(*			
	RAFALOS
	Rafał Osajda		19.09.2025		TC 4024.66
	Element bazowy umożliwiający potomkom wysyłaś zgłoszenia do logera
*)
FUNCTION_BLOCK FB_BaseLoggerElement EXTENDS FB_Base IMPLEMENTS ITF_BaseLoggerElement, ITF_BaseLoggerElement_HMI_Connector
VAR
	itfLogger						: ITF_BaseLogger;
	stIdentifier					: ST_BaseElementIdentifier;
	stEvents						: ST_BaseEvents;
END_VAR

(*			
	EVERDE sp. z o.o.
	Rafał Osajda		24.03.2025		TC 4024.66
	Dodawanie zgłoszenia do systemu
*)
METHOD PUBLIC AddEvent : BOOL
VAR_INPUT
	bIgnoreRepetitions					: BOOL;						//jak true nie zliczaj powtorzeń wystapienia np komunikaty
	eEventCategory						: E_BaseEvents_Category;	//BYTE;	//1 - blad, 2 - ostrzezenie, 3 - wiadomosc, 4 - safety
	bConfirm							: BOOL;						//wymaga powtierdzenia
	stDescription						: ST_BaseLabel;
END_VAR
IF (THIS^.stEvents.uiNumberOfAdded + 1 <= GVL_BaseConstans.MAX_ILOSC_ZGLOSZEN_NA_ELEMENT) THEN
	THIS^.stEvents.uiNumberOfAdded														:= THIS^.stEvents.uiNumberOfAdded + 1;
	THIS^.stEvents.arrDefinitions [THIS^.stEvents.uiNumberOfAdded].uiIDInItem			:= THIS^.stEvents.uiNumberOfAdded;
	THIS^.stEvents.arrDefinitions [THIS^.stEvents.uiNumberOfAdded].bIgnoreRepetitions	:= bIgnoreRepetitions;
	THIS^.stEvents.arrDefinitions [THIS^.stEvents.uiNumberOfAdded].eEventCategory		:= eEventCategory;
	THIS^.stEvents.arrDefinitions [THIS^.stEvents.uiNumberOfAdded].stDescription		:= stDescription;
	THIS^.stEvents.arrDefinitions [THIS^.stEvents.uiNumberOfAdded].bConfirm				:= bConfirm;
	AddEvent						:= TRUE;
ELSE
	AddEvent						:= FALSE;
END_IF
END_METHOD

(*			
	EVERDE sp. z o.o.
	Rafał Osajda		24.03.2025		TC 4024.66
	Definicja nowego zgłoszenia
*)
METHOD PUBLIC EventsDefinition : BOOL
MEMSET (
	destAddr		:= ADR (THIS^.stEvents.arrDefinitions),
	fillByte		:= 0,
	n				:= SIZEOF (THIS^.stEvents.arrDefinitions)
);
THIS^.stEvents.uiNumberOfAdded	:= 0;
END_METHOD

(*			
	RAFALOS
	Rafał Osajda		25.09.2025		TC 4024.66
	Metoda wywoływana w pierwszym cyklu
*)
METHOD PUBLIC FirstCycle : BOOL
VAR_INPUT
END_VAR

FirstCycle				:= TRUE;
END_METHOD

METHOD PUBLIC GetCode : STRING
VAR_INPUT
END_VAR
GetCode			:= THIS^.stIdentifier.sCode;
END_METHOD

METHOD PUBLIC GetID : UINT
VAR_INPUT
END_VAR
GetID				:= THIS^.stIdentifier.uiID;
END_METHOD

METHOD PUBLIC GetIdentyfier : ST_BaseElementIdentifier
VAR_INPUT
END_VAR
GetIdentyfier				:= THIS^.stIdentifier;
END_METHOD

METHOD PUBLIC GetName : ST_BaseLabel
VAR_INPUT
END_VAR
GetName				:= THIS^.stIdentifier.stName;
END_METHOD

METHOD PUBLIC GetType : E_BaseElementType
VAR_INPUT
END_VAR
GetType				:= THIS^.stIdentifier.eType;
END_METHOD

METHOD PUBLIC SetCode
VAR_INPUT
	sCode							: STRING;
END_VAR
THIS^.stIdentifier.sCode				:= sCode;
END_METHOD

METHOD PUBLIC SetID
VAR_INPUT
	uiID					: UINT;
END_VAR
THIS^.stIdentifier.uiID			:= uiID;
END_METHOD

METHOD PUBLIC SetName
VAR_INPUT
	stName				: ST_BaseLabel;
END_VAR
this^.stIdentifier.stName			:= stName;
END_METHOD

METHOD PUBLIC SetType
VAR_INPUT
	eType					: E_BaseElementType;
END_VAR
THIS^.stIdentifier.eType				:= eType;
END_METHOD

END_FUNCTION_BLOCK

(* stored: Version 1.1.0.1
   POU FB_BaseLoggerElement: Id {84ce134f-38cc-08bd-3d60-40e507799b32}, SpecialFunc None
   Folder Events: Id {0a451ccb-a5c6-0466-1fb3-43b9aac577ff}
   Folder ID: Id {9f4accde-c200-0e3a-3280-17fd6d107d51}
   Folder ITF_BaseLoggerElement_HMI_Connector: Id {abdbf241-16b7-0948-3bea-83a764b01a75}
   Method AddEvent: Id {634f9b8e-85a8-02a3-013c-6c409e6a5e93}
   Method EventsDefinition: Id {d570146c-fc2a-0a65-1409-5460668a36c6}
   Method FirstCycle: Id {c59af0fe-9b69-0431-255c-4b5a82a26450}
   Method GetCode: Id {af745aea-1b66-059b-10b2-395e94251847}
   Method GetID: Id {76a78e74-7761-0532-0c6a-49d51d5b5955}
   Method GetIdentyfier: Id {48d63181-6e27-0c5e-3c1d-ae09759ac84b}
   Method GetName: Id {f31b5203-9f85-03eb-3e31-406645634fd5}
   Method GetType: Id {61940ec7-463b-0e69-2135-9287ae34093b}
   Method SetCode: Id {fe7a56f6-55e1-0e90-11d6-90800c0cf084}
   Method SetID: Id {9acba3a6-fc5f-0ece-1ab3-a775104efe88}
   Method SetName: Id {206e85b8-29f8-08fa-23dd-60a3f6071df5}
   Method SetType: Id {bf11665f-1c90-0e8a-0bd5-6357f50d48e0} *)
